{attribute 'qualified_only'}
{attribute 'strict'}
{attribute 'to_string'}
TYPE EMppcCollector :
(
	Unknown := 0,
    WIDE,
    NARROW
);
END_TYPE

(* stored: Version 1.1.0.1, ProductVersion 3.1.4024.12
   DUT EMppcCollector: Id {d0b73c9b-c0d9-4288-ae93-dfcbfa5f7e73} *)
